// TIA Portal V15.1 export
// export: Created 2024-05-17T05:38:59.4629069Z, ExportSetting WithDefaults, DisplayName Totally Integrated Automation Portal, DisplayVersion V15.1 Update 5, DisplayName TIA Portal Openness, DisplayVersion V15.1 Update 5, DisplayName SINAMICS Startdrive Advanced, DisplayVersion V15.1, DisplayName G130, G150, S120, S150, SINAMICS MV, S210, DisplayVersion V15.1, DisplayName G110M, G120, G120C, G120D, G120P, DisplayVersion V15.1, DisplayName STEP 7 Professional, DisplayVersion V15.1 Update 5, DisplayName STEP 7 Safety, DisplayVersion V15.1, DisplayName WinCC Professional, DisplayVersion V15.1 Update 5, DisplayName SIMATIC Visualization Architect, DisplayVersion V15.1
FUNCTION "209000NCP01PNIODiagList" : Void   // FC271, FBD
TITLE = 0118100PNIODiagList / 209000NCP01PNIODiagList
{ S7_Optimized_Access := 'TRUE' }
VERSION : 0.1
// stored: AutoNumber false, IsIECCheckEnabled false, SetENOAutomatically False, UDAEnableTagReadback false
   VAR_TEMP   // added for the SCL form of the ladder/FBD networks
      _w1 : Bool;
      _w2 : Bool;
   END_VAR
BEGIN

REGION Network 1: **** 3.1 - Communication - Other Systems **** PN-Diag S7-15xxF -- List with IP adress
   // List with IP adress
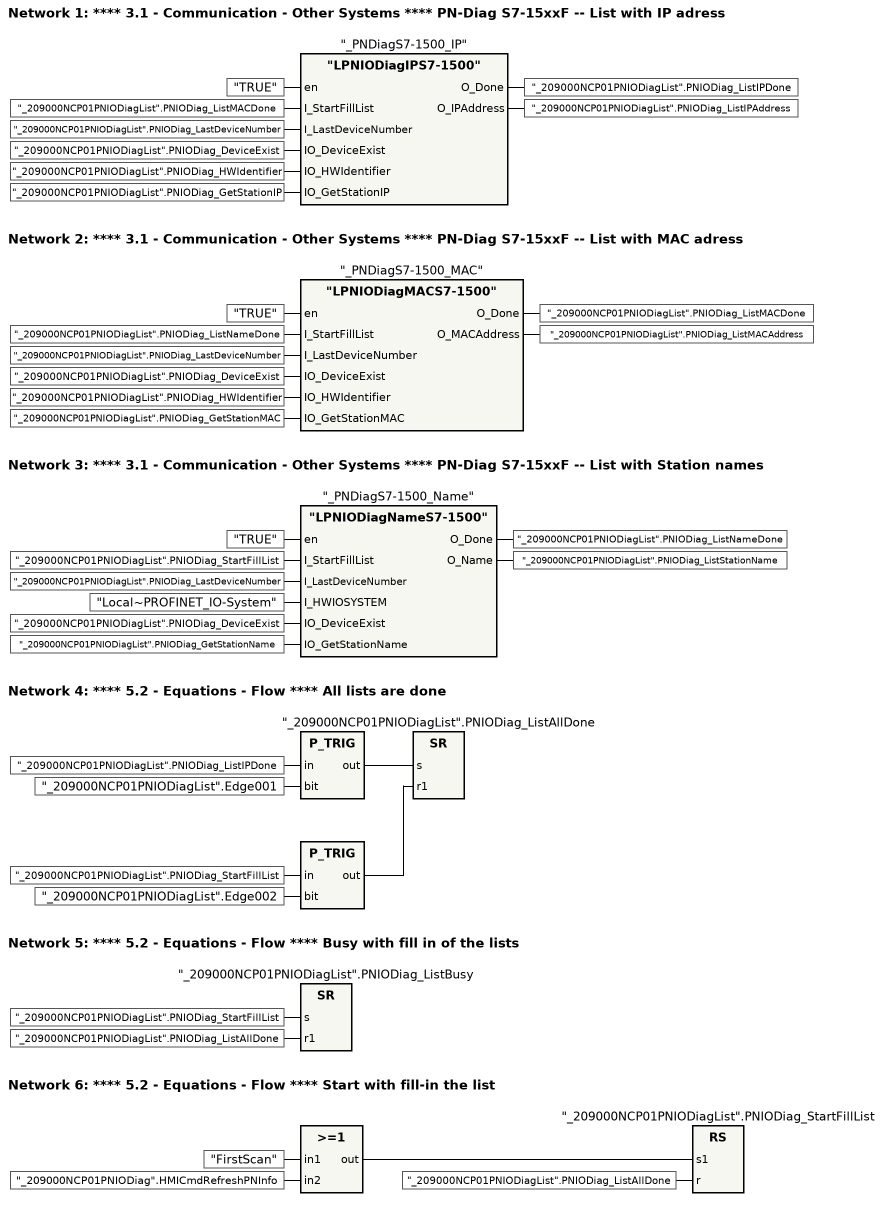
   IF "TRUE" THEN
       "_PNDiagS7-1500_IP"(I_StartFillList := "_209000NCP01PNIODiagList".PNIODiag_ListMACDone,   // "LPNIODiagIPS7-1500"
                           I_LastDeviceNumber := "_209000NCP01PNIODiagList".PNIODiag_LastDeviceNumber,
                           IO_DeviceExist := "_209000NCP01PNIODiagList".PNIODiag_DeviceExist,
                           IO_HWIdentifier := "_209000NCP01PNIODiagList".PNIODiag_HWIdentifier,
                           IO_GetStationIP := "_209000NCP01PNIODiagList".PNIODiag_GetStationIP,
                           O_Done => "_209000NCP01PNIODiagList".PNIODiag_ListIPDone,
                           O_IPAddress => "_209000NCP01PNIODiagList".PNIODiag_ListIPAddress);
   END_IF;
END_REGION

REGION Network 2: **** 3.1 - Communication - Other Systems **** PN-Diag S7-15xxF -- List with MAC adress
   // List with MAC adress
   IF "TRUE" THEN
       "_PNDiagS7-1500_MAC"(I_StartFillList := "_209000NCP01PNIODiagList".PNIODiag_ListNameDone,   // "LPNIODiagMACS7-1500"
                            I_LastDeviceNumber := "_209000NCP01PNIODiagList".PNIODiag_LastDeviceNumber,
                            IO_DeviceExist := "_209000NCP01PNIODiagList".PNIODiag_DeviceExist,
                            IO_HWIdentifier := "_209000NCP01PNIODiagList".PNIODiag_HWIdentifier,
                            IO_GetStationMAC := "_209000NCP01PNIODiagList".PNIODiag_GetStationMAC,
                            O_Done => "_209000NCP01PNIODiagList".PNIODiag_ListMACDone,
                            O_MACAddress => "_209000NCP01PNIODiagList".PNIODiag_ListMACAddress);
   END_IF;
END_REGION

REGION Network 3: **** 3.1 - Communication - Other Systems **** PN-Diag S7-15xxF -- List with Station names
   // List with Station names
   IF "TRUE" THEN
       "_PNDiagS7-1500_Name"(I_StartFillList := "_209000NCP01PNIODiagList".PNIODiag_StartFillList,   // "LPNIODiagNameS7-1500"
                             I_LastDeviceNumber := "_209000NCP01PNIODiagList".PNIODiag_LastDeviceNumber,
                             I_HWIOSYSTEM := "Local~PROFINET_IO-System",
                             IO_DeviceExist := "_209000NCP01PNIODiagList".PNIODiag_DeviceExist,
                             IO_GetStationName := "_209000NCP01PNIODiagList".PNIODiag_GetStationName,
                             O_Done => "_209000NCP01PNIODiagList".PNIODiag_ListNameDone,
                             O_Name => "_209000NCP01PNIODiagList".PNIODiag_ListStationName);
   END_IF;
END_REGION

REGION Network 4: **** 5.2 - Equations - Flow **** All lists are done
   // All lists are done
   #_w1 := "_209000NCP01PNIODiagList".PNIODiag_ListIPDone AND NOT "_209000NCP01PNIODiagList".Edge001;   // rising edge
   "_209000NCP01PNIODiagList".Edge001 := "_209000NCP01PNIODiagList".PNIODiag_ListIPDone;
   #_w2 := "_209000NCP01PNIODiagList".PNIODiag_StartFillList AND NOT "_209000NCP01PNIODiagList".Edge002;   // rising edge
   "_209000NCP01PNIODiagList".Edge002 := "_209000NCP01PNIODiagList".PNIODiag_StartFillList;
   IF #_w1 THEN
       "_209000NCP01PNIODiagList".PNIODiag_ListAllDone := TRUE;   // SR flip-flop
   END_IF;
   IF #_w2 THEN "_209000NCP01PNIODiagList".PNIODiag_ListAllDone := FALSE; END_IF;
END_REGION

REGION Network 5: **** 5.2 - Equations - Flow **** Busy with fill in of the lists
   // Busy with fill in of the lists
   IF "_209000NCP01PNIODiagList".PNIODiag_StartFillList THEN
       "_209000NCP01PNIODiagList".PNIODiag_ListBusy := TRUE;   // SR flip-flop
   END_IF;
   IF "_209000NCP01PNIODiagList".PNIODiag_ListAllDone THEN
       "_209000NCP01PNIODiagList".PNIODiag_ListBusy := FALSE;
   END_IF;
END_REGION

REGION Network 6: **** 5.2 - Equations - Flow **** Start with fill-in the list
   // Start with fill-in the list
   IF "_209000NCP01PNIODiagList".PNIODiag_ListAllDone THEN
       "_209000NCP01PNIODiagList".PNIODiag_StartFillList := FALSE;   // RS flip-flop
   END_IF;
   IF "FirstScan" OR "_209000NCP01PNIODiag".HMICmdRefreshPNInfo THEN
       "_209000NCP01PNIODiagList".PNIODiag_StartFillList := TRUE;
   END_IF;
END_REGION
END_FUNCTION
